// Mitsubishi GX Works2 project: msp_3   PLC: Q03UDV

PROGRAM MAIN
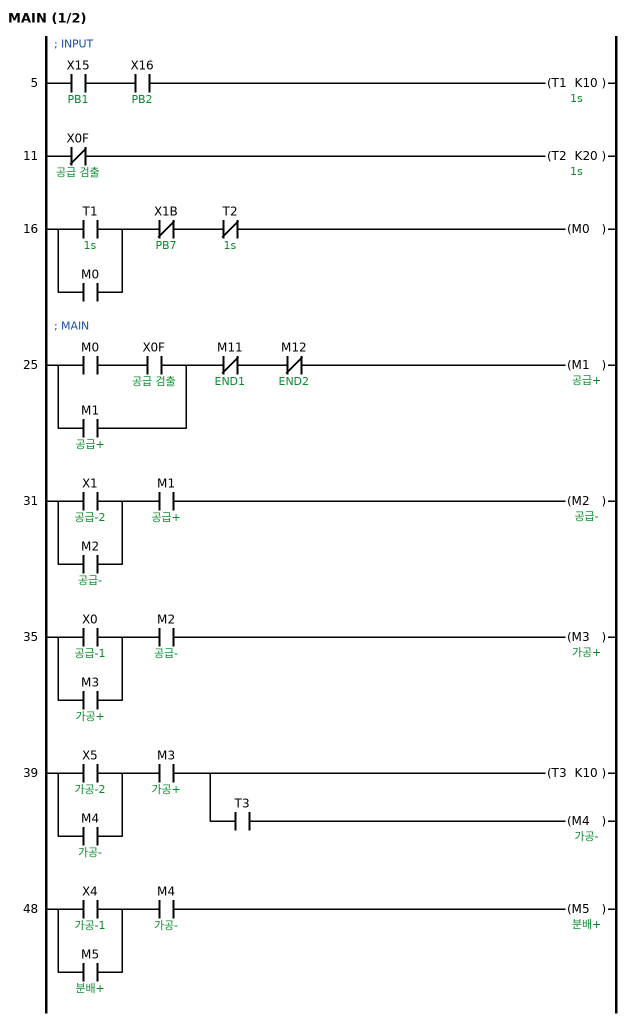
; INPUT
5     LD      X15  ; PB1
      AND     X16  ; PB2
      OUT     T1 K10  ; 1s
11    LDI     X0F  ; 공급 검출
      OUT     T2 K20  ; 1s
16    LD      T1  ; 1s
      OR      M0
      ANI     X1B  ; PB7
      ANI     T2  ; 1s
      OUT     M0
; MAIN
25    LD      M0
      AND     X0F  ; 공급 검출
      OR      M1  ; 공급+
      ANI     M11  ; END1
      ANI     M12  ; END2
      OUT     M1  ; 공급+
31    LD      X1  ; 공급-2
      OR      M2  ; 공급-
      AND     M1  ; 공급+
      OUT     M2  ; 공급-
35    LD      X0  ; 공급-1
      OR      M3  ; 가공+
      AND     M2  ; 공급-
      OUT     M3  ; 가공+
39    LD      X5  ; 가공-2
      OR      M4  ; 가공-
      AND     M3  ; 가공+
      OUT     T3 K10
      AND     T3
      OUT     M4  ; 가공-
48    LD      X4  ; 가공-1
      OR      M5  ; 분배+
      AND     M4  ; 가공-
      OUT     M5  ; 분배+
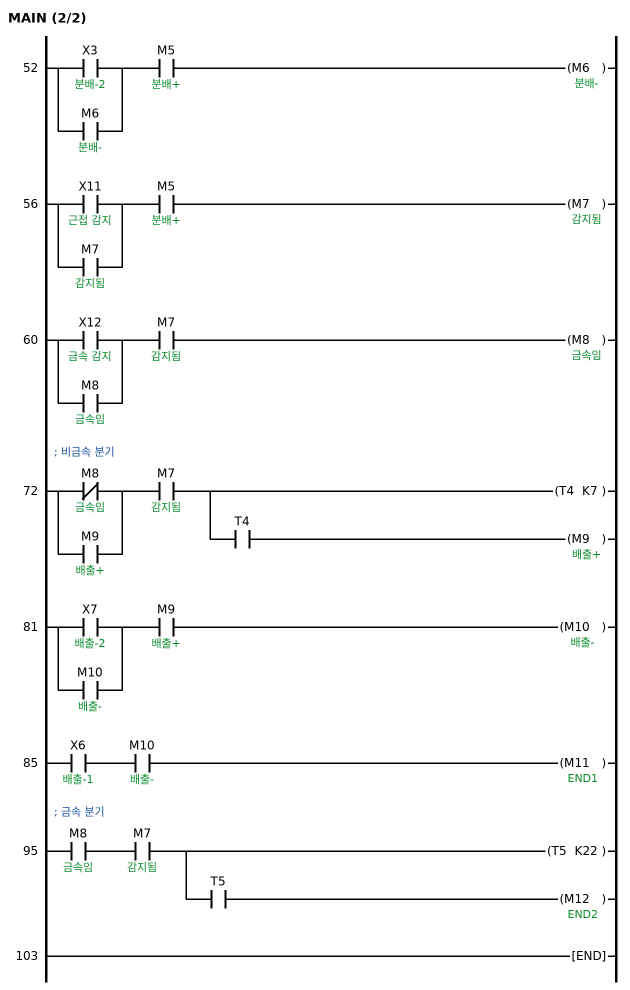
52    LD      X3  ; 분배-2
      OR      M6  ; 분배-
      AND     M5  ; 분배+
      OUT     M6  ; 분배-
56    LD      X11  ; 근접 감지
      OR      M7  ; 감지됨
      AND     M5  ; 분배+
      OUT     M7  ; 감지됨
60    LD      X12  ; 금속 감지
      OR      M8  ; 금속임
      AND     M7  ; 감지됨
      OUT     M8  ; 금속임
; 비금속 분기
72    LDI     M8  ; 금속임
      OR      M9  ; 배출+
      AND     M7  ; 감지됨
      OUT     T4 K7
      AND     T4
      OUT     M9  ; 배출+
81    LD      X7  ; 배출-2
      OR      M10  ; 배출-
      AND     M9  ; 배출+
      OUT     M10  ; 배출-
85    LD      X6  ; 배출-1
      AND     M10  ; 배출-
      OUT     M11  ; END1
; 금속 분기
95    LD      M8  ; 금속임
      AND     M7  ; 감지됨
      OUT     T5 K22
      AND     T5
      OUT     M12  ; END2
103   END
END_PROGRAM

PROGRAM OUTPUT
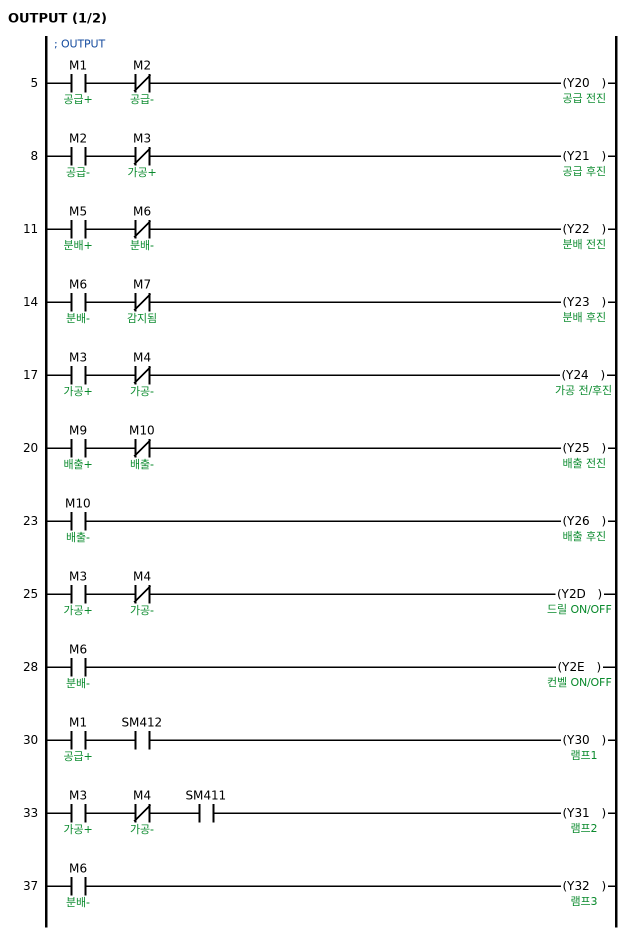
; OUTPUT
5     LD      M1  ; 공급+
      ANI     M2  ; 공급-
      OUT     Y20  ; 공급 전진
8     LD      M2  ; 공급-
      ANI     M3  ; 가공+
      OUT     Y21  ; 공급 후진
11    LD      M5  ; 분배+
      ANI     M6  ; 분배-
      OUT     Y22  ; 분배 전진
14    LD      M6  ; 분배-
      ANI     M7  ; 감지됨
      OUT     Y23  ; 분배 후진
17    LD      M3  ; 가공+
      ANI     M4  ; 가공-
      OUT     Y24  ; 가공 전/후진
20    LD      M9  ; 배출+
      ANI     M10  ; 배출-
      OUT     Y25  ; 배출 전진
23    LD      M10  ; 배출-
      OUT     Y26  ; 배출 후진
25    LD      M3  ; 가공+
      ANI     M4  ; 가공-
      OUT     Y2D  ; 드릴 ON/OFF
28    LD      M6  ; 분배-
      OUT     Y2E  ; 컨벨 ON/OFF
30    LD      M1  ; 공급+
      AND     SM412
      OUT     Y30  ; 램프1
33    LD      M3  ; 가공+
      ANI     M4  ; 가공-
      AND     SM411
      OUT     Y31  ; 램프2
37    LD      M6  ; 분배-
      OUT     Y32  ; 램프3
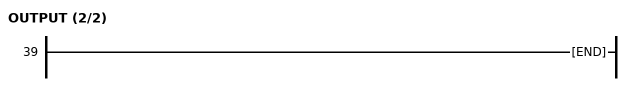
39    END
END_PROGRAM

// device comments not shown above
X2  ; 분배-1
X8  ; 스토퍼-1
X9  ; 스토퍼-2
X0A  ; 흡착-1
X0B  ; 흡착-2
X0C  ; 흡착 검출
X0D  ; 창고-1
X0E  ; 창고-2
X10  ; 공급 검출
X13  ; 스토퍼 감지
X14  ; 컨벨 인코더
X17  ; PB3
X18  ; PB4
X19  ; PB5
X1A  ; PB6
X1C  ; PB8
X20  ; A 전진
X21  ; A 후진
X24  ; B 전진/후진
X2D  ; 가공 모터
Y27  ; 스토퍼 전/후진
Y28  ; 흡착 전진
Y29  ; 흡착 후진
Y2A  ; 흡착 ON/OFF
Y2B  ; 창고 전진
Y2C  ; 창고 후진
Y33  ; 램프4
Y34  ; 램프5
Y35  ; 램프6
Y36  ; 램프7
Y37  ; 부저
